{attribute 'GeneratedUsingTerminal: EK1100-0000-0018'}
{attribute addProperty BoxType "EK1100-0000-0018"}
{attribute addProperty Id "Beckhoff_EJ6xxxEK1122Beckhoff_EJ6xxxEK1122_737473AE2A_0001_EJ6002_0000_0016EJ6002_D5B468BD126A_0002_EJ6224_0000_0016EJ6224_98EF241924A_0003_EJ6224_0090_0016EJ6224_98EF241924"}
{attribute addProperty CRC "3548435934"}
{attribute addProperty Size "176"}
TYPE Beckhoff_EJ6xxx_D380D5DE EXTENDS EK1100_1FC0878B :
STRUCT
	{attribute addProperty Name "Beckhoff_EJ6xxxEK1122"}
	{attribute addProperty PreviousPort "Beckhoff EJ6xxx : B"}
	Beckhoff_EJ6xxxEK1122 : Beckhoff_EJ6xxxEK1122_737473AE;
	{attribute addProperty Name "A_0001_EJ6002_0000_0016"}
	{attribute addProperty PreviousPort "Beckhoff EJ6xxxEK1122 : C"}
	A_0001_EJ6002_0000_0016 : EJ6002_D5B468BD;
	{attribute addProperty Name "A_0002_EJ6224_0000_0016"}
	{attribute addProperty PreviousPort "A_0001(EJ6002-0000-0016) : B"}
	A_0002_EJ6224_0000_0016 : EJ6224_98EF2419;
	{attribute addProperty Name "A_0003_EJ6224_0090_0016"}
	{attribute addProperty PreviousPort "A_0002(EJ6224-0000-0016) : B"}
	A_0003_EJ6224_0090_0016 : EJ6224_98EF2419;
END_STRUCT
END_TYPE

(* stored: Version 1.2.0.0, ProductVersion 3.1.4024.9
   DUT Beckhoff_EJ6xxx_D380D5DE: Id {ad700bb5-bb16-4f0b-8de9-7a225d42ddc0} *)
